(* CoDeSys 2.3 export: EXTRACT.EXP *)

(* POU bit/byte functions/EXTRACT, ST *)
(* function returns Bit N of value X *)
FUNCTION EXTRACT : BOOL
VAR_INPUT
	X:DWORD;	(* value *)
	N:BYTE;		(* number of bit to be extracted *)
END_VAR
VAR
END_VAR
(* @TEXT_IMPLEMENTATION := 'ST' *)
EXTRACT:=((SHR(X,N) AND 1)=1);
END_FUNCTION
